{attribute 'qualified_only'}
{attribute 'strict'}
{attribute 'to_string'}
TYPE E_Type :
(
	alarm := 0,
	message := 1
);
END_TYPE

(* stored: Version 1.1.0.1, ProductVersion 3.1.4024.9
   DUT E_Type: Id {1831786b-cc3b-4584-a83b-58839ae4003a} *)
